FUNCTION_BLOCK FB_Keba_keypad_tcp
VAR_INPUT
END_VAR
VAR_OUTPUT
END_VAR
VAR

	fbSocketCloseAll	:FB_SocketCloseAll;
	xStartup			: BOOL := TRUE;
	myServer			: T_HSERVER;
	
	server 				: FB_ServerClientConnection;
	xEnable				: BOOL := FALSE;
	
	tcp_rec				: FB_SocketReceive;
	xExecute 			: BOOL;
	ton_read			: TON;
	
	dest				: ARRAY[1..1024] OF BYTE;
	myString			: STRING(20);
	
END_VAR
VAR CONSTANT
	AMS_NET			: T_AmsNetID := '192.168.20.200.1.1';
	REC_ARR_SIZE	: UDINT	:= 1024;
END_VAR


IF xStartup THEN (*On PLC reset or program download close all old connections *)
	fbSocketCloseAll( sSrvNetId:= '', bExecute:= TRUE, tTimeout:= T#10S );
ELSE
	fbSocketCloseAll( bExecute:= FALSE );
END_IF	

F_CreateServerHnd(		sSrvNetID := '',
						sLocalHost := '192.168.21.200',
						nLocalPort := 2020,
						nMode := LISTEN_MODE_CLOSEALL,
						bEnable := TRUE,
						hServer := myServer);


server(		hServer := myServer,
			eMode := E_SocketAcceptMode.eACCEPT_SEL_HOST,
			sRemoteHost := '192.168.21.201',
			nRemotePort := 0,
			bEnable := xEnable,
			tReconnect := T#1S);

ton_read(IN := NOT ton_read.Q, PT := T#50MS);
tcp_rec(	sSrvNetId := '',
			hSocket := server.hSocket,
			cbLen := 1024,
			pDest := ADR(dest),
			bExecute := ton_read.Q,
			tTimeout := T#100MS);
			
IF tcp_rec.nRecBytes <> 0 THEN
	STRNCPY(ADR(myString), ADR(dest), 20);
END_IF

xExecute := FALSE;
xStartup := FALSE;

END_FUNCTION_BLOCK

(* stored: Version 1.1.0.1, ProductVersion 3.1.4024.6
   POU FB_Keba_keypad_tcp: Id {aa81aac2-4e75-4757-9515-2eae602c7105}, SpecialFunc None *)
